FUNCTION_BLOCK F_MOD (* modulo *)
  PACKAGE iec61131::arithmetic;
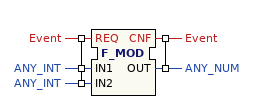
  EVENT_INPUT
    REQ WITH IN1, IN2; (* Normal Execution Request *)
  END_EVENT
  EVENT_OUTPUT
    CNF WITH OUT; (* Execution Confirmation *)
  END_EVENT
  VAR_INPUT
    IN1 : ANY_INT; (* divident input *)
    IN2 : ANY_INT; (* divisor input *)
  END_VAR
  VAR_OUTPUT
    OUT : ANY_NUM; (* rest of IN1 devided by IN2 *)
  END_VAR
END_FUNCTION_BLOCK
